PROGRAM Axe_01_X (*Chariot*)
VAR	
		XChariot: FB_Axe_Ethercat_V2;		
		Defaut_Var_Chariot_AX5000: BOOL;
		Diag_Nbrs_Var_Chariot_AX5000 :UDINT;
		Diag_Mess_Var_Chariot_AX5000: STRING;
END_VAR
VAR // added by the converter: edge detectors and wires of the graphical bodies
    _rt1 : R_TRIG;
END_VAR

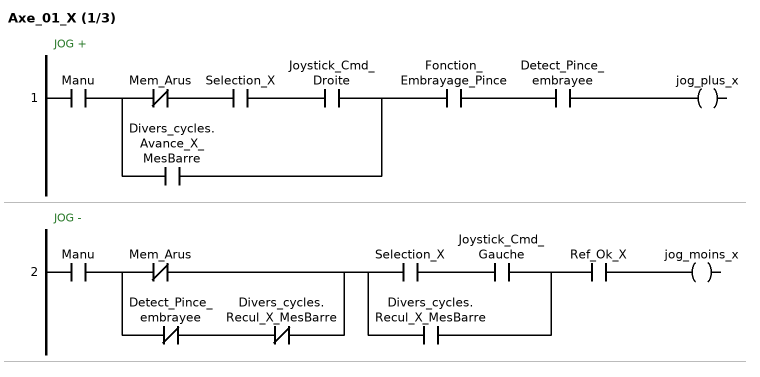
// NETWORK 1
// JOG +
jog_plus_x := Manu AND (NOT Mem_Arus AND Selection_X AND Joystick_Cmd_Droite OR Divers_cycles.Avance_X_MesBarre) AND Fonction_Embrayage_Pince AND Detect_Pince_embrayee;

// NETWORK 2
// JOG -
jog_moins_x := Manu AND (NOT Mem_Arus OR NOT Detect_Pince_embrayee AND NOT Divers_cycles.Recul_X_MesBarre) AND (Selection_X AND Joystick_Cmd_Gauche OR Divers_cycles.Recul_X_MesBarre) AND Ref_Ok_X;

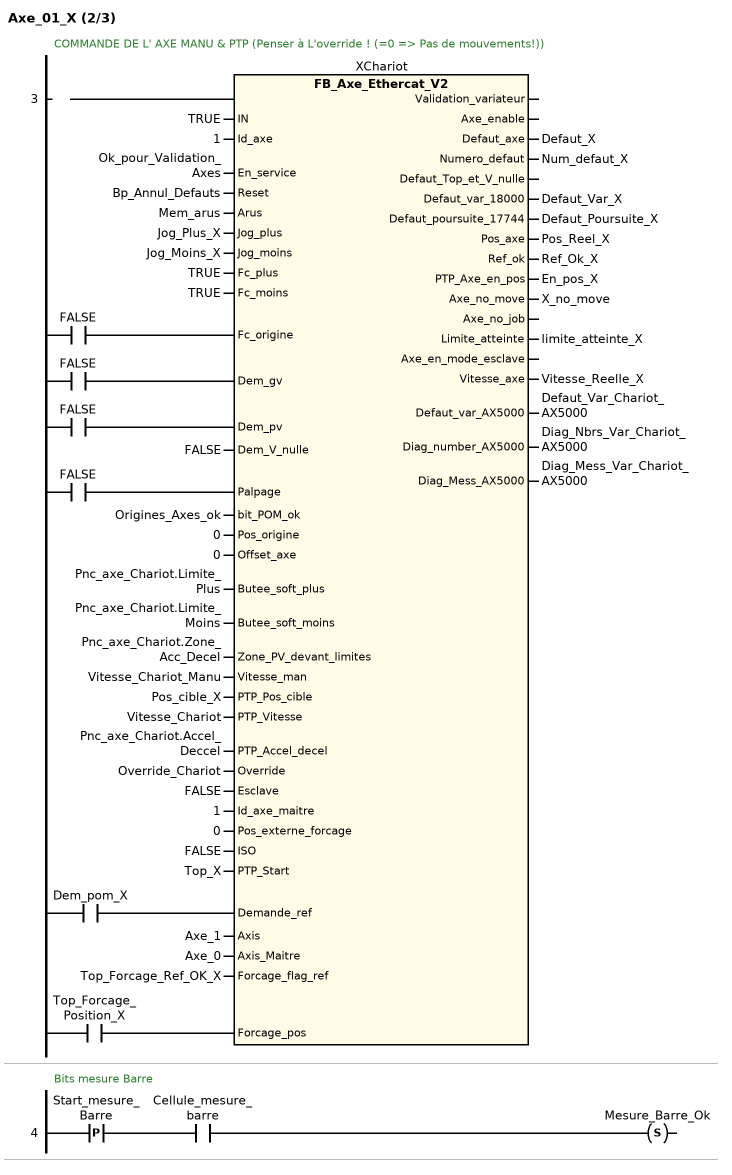
// NETWORK 3
// 					COMMANDE DE L' AXE MANU & PTP (Penser à L'override ! (=0 => Pas de mouvements!))
//
//
XChariot(
    IN := TRUE,
    Id_axe := 1,
    En_service := Ok_pour_Validation_Axes,
    Reset := Bp_Annul_Defauts,
    Arus := Mem_arus,
    Jog_plus := Jog_Plus_X,
    Jog_moins := Jog_Moins_X,
    Fc_plus := TRUE,
    Fc_moins := TRUE,
    Fc_origine := FALSE,
    Dem_gv := FALSE,
    Dem_pv := FALSE,
    Dem_V_nulle := FALSE,
    Palpage := FALSE,
    bit_POM_ok := Origines_Axes_ok,
    Pos_origine := 0,
    Offset_axe := 0,
    Butee_soft_plus := Pnc_axe_Chariot.Limite_Plus,
    Butee_soft_moins := Pnc_axe_Chariot.Limite_Moins,
    Zone_PV_devant_limites := Pnc_axe_Chariot.Zone_Acc_Decel,
    Vitesse_man := Vitesse_Chariot_Manu,
    PTP_Pos_cible := Pos_cible_X,
    PTP_Vitesse := Vitesse_Chariot,
    PTP_Accel_decel := Pnc_axe_Chariot.Accel_Deccel,
    Override := Override_Chariot,
    Esclave := FALSE,
    Id_axe_maitre := 1,
    Pos_externe_forcage := 0,
    ISO := FALSE,
    PTP_Start := Top_X,
    Demande_ref := Dem_pom_X,
    Axis := Axe_1,
    Axis_Maitre := Axe_0,
    Forcage_flag_ref := Top_Forcage_Ref_OK_X,
    Forcage_pos := Top_Forcage_Position_X,
    Defaut_axe => Defaut_X,
    Numero_defaut => Num_defaut_X,
    Defaut_var_18000 => Defaut_Var_X,
    Defaut_poursuite_17744 => Defaut_Poursuite_X,
    Pos_axe => Pos_Reel_X,
    Ref_ok => Ref_Ok_X,
    PTP_Axe_en_pos => En_pos_X,
    Axe_no_move => X_no_move,
    Limite_atteinte => limite_atteinte_X,
    Vitesse_axe => Vitesse_Reelle_X,
    Defaut_var_AX5000 => Defaut_Var_Chariot_AX5000,
    Diag_number_AX5000 => Diag_Nbrs_Var_Chariot_AX5000,
    Diag_Mess_AX5000 => Diag_Mess_Var_Chariot_AX5000); // FB_Axe_Ethercat_V2

// NETWORK 4
// Bits mesure Barre
_rt1(CLK := Start_mesure_Barre);
Mesure_Barre_Ok S= _rt1.Q AND Cellule_mesure_barre;

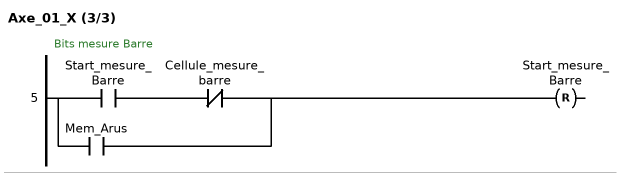
// NETWORK 5
// Bits mesure Barre
Start_mesure_Barre R= Start_mesure_Barre AND NOT Cellule_mesure_barre OR Mem_Arus;

END_PROGRAM

(* stored: Version 1.1.0.1, ProductVersion 3.1.4024.15
   POU Axe_01_X: Id {a4e3e69c-6c89-4434-b00d-143c546b94c4}, SpecialFunc None *)
